TYPE "Prod_Beam_Area"
VERSION : 0.1
// Block: Prod_Beam_Area
   STRUCT
      Halted : Prod_Halted;
      Man : Bool;
      Doors_Closed : Bool;
      CycleON : Bool;
      Running : Bool;
      SetUpDone : Bool;
      SetupDone_Ax : Array[1..9] of Bool;
   END_STRUCT;

END_TYPE
